FUNCTION_BLOCK FINAL IsJsonMemberString IMPLEMENTS Callback
VAR_INPUT
	jsonDomParser: REFERENCE TO FB_JsonDomParser;
	memberReference: REFERENCE TO SJsonValue;
	isStringReference: REFERENCE TO BOOL;
END_VAR

(* This is method get's exectued by the framework when the callback is triggered.
 It returns a step number which might be used together with Await to jump to a certain chain step
 after the callback code has been executed.*)
METHOD execute : UDINT
isStringReference := memberReference <> 0 AND_THEN jsonDomParser.IsString(memberReference);
END_METHOD

END_FUNCTION_BLOCK

(* stored: Version 1.1.0.1, ProductVersion 3.1.4024.12
   POU IsJsonMemberString: Id {cefea03f-a64a-48bf-8b03-1bc2207323cb}, SpecialFunc None
   Method execute: Id {a929a389-e58e-4615-a817-a1eab03a5f46} *)
